PROGRAM MAIN
VAR
	test: BOOL;

END_VAR

F_FactoryIO_Read_Inputs();
F_FactoryIO_Read_InputRegs();
F_FactoryIO_Write_Coils();
F_FactoryIO_WriteRegs();

test := GAB_FactoryIO_Inputs[0].0;

END_PROGRAM

(* stored: Version 1.1.0.1, ProductVersion 3.1.4024.11
   POU MAIN: Id {11a895ac-5a06-4334-87ae-34581a64c27e}, SpecialFunc None *)
